{attribute 'linkalways'} 
{attribute 'no_explicit_call' := 'This FB is a CLASS and must be accessed using methods or properties'}
{attribute 'enable_dynamic_creation'}
FUNCTION_BLOCK MockDatatype_BOOL EXTENDS DatatypeBase
VAR
	localData : BOOL;
	activeData : REFERENCE TO BOOL REF= localData;
END_VAR

PROPERTY PUBLIC Address : PVOID
GET
Address := ADR(activeData);
END_GET
END_PROPERTY

METHOD PUBLIC ClearReference
VAR_INPUT
END_VAR
activeData REF= localData;
END_METHOD

METHOD PUBLIC Clone : I_Datatype
VAR
    pClone : POINTER TO MockDatatype_BOOL;
END_VAR
pClone := __NEW(MockDatatype_BOOL(InitialValue := Value));
Clone := pClone^;
END_METHOD

METHOD FB_init : BOOL
VAR_INPUT
	bInitRetains : BOOL; // if TRUE, the retain variables are initialized (warm start / cold start)
	bInCopyCode : BOOL;  // if TRUE, the instance afterwards gets moved into the copy code (online change)
	InitialValue : BOOL;
END_VAR
localData := InitialValue;
END_METHOD

METHOD PUBLIC MakeReferenceTo
VAR_INPUT
	ReferenceTarget : REFERENCE TO BOOL;
END_VAR
activeData REF= ReferenceTarget;
END_METHOD

METHOD PUBLIC SerializeWith
VAR_INPUT
	Serializer : I_Serializer;
END_VAR
Serializer.AddBool(activeData);
END_METHOD

PROPERTY PUBLIC Size : UDINT
GET
Size := SIZEOF(activeData);
END_GET
END_PROPERTY

METHOD TryDeserializeFrom : BOOL
VAR_INPUT
	Deserializer : I_Deserializer;
	Feedback : I_DeserializerFeedback;
END_VAR
TryDeserializeFrom := Deserializer.TryGetBool(activeData, Feedback);
END_METHOD

METHOD TryMakeReferenceTo : BOOL
VAR_INPUT
	Target : I_Datatype;
END_VAR
VAR
	pTargetData : POINTER TO BOOL;
END_VAR
IF NOT (Target.TypeName = TypeName) THEN
	RETURN;
END_IF

pTargetData := Target.Address;
activeData REF= pTargetData^;
TryMakeReferenceTo := TRUE;
END_METHOD

PROPERTY PUBLIC TypeName : T_MAXSTRING
GET
TypeName := 'BOOL';
END_GET
END_PROPERTY

PROPERTY PUBLIC Value : BOOL
GET
Value := activeData;
END_GET
SET
activeData := Value;
END_SET
END_PROPERTY

END_FUNCTION_BLOCK

(* stored: Version 1.1.0.1, ProductVersion 3.1.4024.12
   POU MockDatatype_BOOL: Id {d86b57f3-7abc-4274-ae09-e4159b41fdfc}, SpecialFunc None
   Folder Constructor: Id {70dfba46-4ea8-44c3-87e2-59949dbe5ffa}
   Property Address: Id {4bca5794-4d5d-430e-8518-b7fcea23a642}
   Get Get: Id {0b080db4-a33e-478d-93f6-5efcf78453a0}
   Method ClearReference: Id {7c34fa36-e620-4f84-964c-c92246c1a6ba}
   Method Clone: Id {f10aea8c-11f7-46d5-8126-275c28ae21df}
   Method FB_init: Id {bb3246cb-9522-473f-9a41-72fd8a1177a7}
   Method MakeReferenceTo: Id {0c9cd5c8-7466-49d9-b7e9-f01eb69bb472}
   Method SerializeWith: Id {1b83739f-9aa1-4545-874d-d72d5ca46bae}
   Property Size: Id {5d01c6d3-3aca-42db-bad6-c0d53c8b2a50}
   Get Get: Id {819358d0-fe15-4ac7-80eb-342c3f84802f}
   Method TryDeserializeFrom: Id {a9b4aa66-ac10-4f97-b0b4-3a3853e8ae9d}
   Method TryMakeReferenceTo: Id {c8eea0ca-4c90-4a2d-a147-5dd9aac9182f}
   Property TypeName: Id {eb827a17-b560-452a-ad90-accac71a0197}
   Get Get: Id {f3069bb3-1217-4d7b-bd58-a9504a904ec1}
   Property Value: Id {9c36f494-b1cb-49a7-903e-f0dda2a5a724}
   Get Get: Id {feebd140-9c42-4c21-a754-6e54d04bd79d}
   Set Set: Id {08c57b1c-cff9-4079-b74c-47800bd08bd7} *)
